// TwinCAT 3 PLC project MainPlc
// ProgramVersion: 3.1.4023.0
// libraries:
//   Tc2_Standard, * (Beckhoff Automation GmbH)
//   Tc2_System, * (Beckhoff Automation GmbH)
//   Tc3_Module, * (Beckhoff Automation GmbH)
// project tree:
//   App/Components/ fbDigitalSensor.TcPOU, fbPneumaticActuator.TcPOU, fbStepConveyor.TcPOU, stComponents.TcDUT, stPneumatics.TcDUT
//   App/Data/ fcEvalConitinuos.TcPOU, stContinuosValueData.TcDUT, stData.TcDUT
//   App/ enumMode.TcDUT (not stored), fbStation.TcPOU, MAIN.TcPOU
//   / IO.TcGVL, PlcTask.TcTTO (not stored)
//   ValueSimulation/ fbValueSimulation.TcPOU
// real-time tasks:
//   TASK PlcTask: cycle T#10ms, priority 20, ADS port 350
// I/O:
//   DEVICE Device 1 (EtherCAT) (disabled), AmsNetId 172.20.10.235.2.1
//     Term 1 (EK1100) [EK1100 EtherCAT Coupler (2A E-Bus)]
//       10A1 (EL1809) [EL1809 16Ch. Dig. Input 24V, 3ms]
//       10A2 (EL2809) [EL2809 16Ch. Dig. Output 24V, 0.5A]
// variable links:
//   MainPlc/MainPlc Instance <-> Device 1 (EtherCAT)/Term 1 (EK1100)/10A1 (EL1809)
//     PlcTask Inputs/IO.i10A1_CH{1..16} <-> Channel {1..16}/Input  (16 links)
//   MainPlc/MainPlc Instance <-> Device 1 (EtherCAT)/Term 1 (EK1100)/10A2 (EL2809)
//     PlcTask Outputs/IO.q10A2_CH{1..16} <-> Channel {1..16}/Output  (16 links)

// ---- App/Components/stComponents.TcDUT
{attribute wpf [Container(Layout.Tabs)]}
{attribute addProperty Name "<#Components#>"}
TYPE stComponents :
STRUCT		
	_pneumatics : stPneumatics;
	{attribute addProperty Name "<#Input step conveyor#> A4"}
	_inputConveyor : fbStepConveyor;	
	{attribute addProperty Name "<#Brick in the take-off position#>"}
	_BrickInTakeOffPosition : fbDigitalSensor;
	{attribute addProperty Name "<#Brick in the gripper#>"}
	_BrickInGripper : fbDigitalSensor;
	{attribute wpf [Container(Layout.Stack, "Measurement sensors")]}
	{attribute addProperty Name "<#Sensor dim X#>"}
	_X_DimSensor : REAL;
	{attribute addProperty Name "<#Sensor dim Y#>"}
	_Y_DimSensor : REAL;
	{attribute addProperty Name "<#Sensor dim Z#>"}
	_Z_DimSensor : REAL;
END_STRUCT
END_TYPE

// ---- App/Components/stPneumatics.TcDUT
{attribute wpf [Container(Layout.Stack)]}
{attribute addProperty Name "<#Pneumatics#>"}
TYPE stPneumatics :
STRUCT
	{attribute addProperty Name "<#Horizontal piston#> A1"}	
	_horizontalPiston : fbPneumaticActuator;
	{attribute addProperty Name "<#Vertical piston#> A2"}
	_verticalPiston : fbPneumaticActuator;
	{attribute addProperty Name "<#Gripper#> A3"}
	_gripper : fbPneumaticActuator;
	{attribute addProperty Name "<#Input end conveyor stopper#> A4"}
	_conveyorEndStopper : fbPneumaticActuator;		
END_STRUCT
END_TYPE

// ---- App/Data/stContinuosValueData.TcDUT
{attribute wpf [Container(Layout.Wrap)]}
{attribute wpf [Group(Layout.GroupBox)]}
TYPE stContinuosValueData :
STRUCT
	{attribute addProperty Name "<#Min#>"}
	Mininum : REAL;
	{attribute wpf [RenderIgnore("Control", "ShadowControl")]}
	{attribute addProperty Name "<#Aquired#>"}	
	Measured : REAL;
	{attribute addProperty Name "<#Max#>"}
	Maximum : REAL;	
END_STRUCT
END_TYPE

// ---- App/Data/stData.TcDUT
{attribute wpf [Container(Layout.Stack)]}
TYPE stData :
STRUCT
	{attribute addProperty Name "<#DimensionX#> [mm]"}			
	DimX : stContinuosValueData;
	{attribute addProperty Name "<#DimensionY#> [mm]"}
	DimY : stContinuosValueData;
	{attribute addProperty Name "<#DimensionZ#> [mm]"}
	DimZ : stContinuosValueData;
END_STRUCT
END_TYPE

// ---- IO.TcGVL
{attribute 'qualified_only'}
VAR_GLOBAL
	i10A1_CH1	AT %I* :BOOL;
	i10A1_CH2	AT %I* :BOOL;
	i10A1_CH3	AT %I* :BOOL;
	i10A1_CH4	AT %I* :BOOL;
	i10A1_CH5	AT %I* :BOOL;
	i10A1_CH6	AT %I* :BOOL;
	i10A1_CH7	AT %I* :BOOL;
	i10A1_CH8	AT %I* :BOOL;
	i10A1_CH9	AT %I* :BOOL;
	i10A1_CH10	AT %I* :BOOL;
	i10A1_CH11	AT %I* :BOOL;
	i10A1_CH12	AT %I* :BOOL;
	i10A1_CH13	AT %I* :BOOL;
	i10A1_CH14	AT %I* :BOOL;
	i10A1_CH15	AT %I* :BOOL;
	i10A1_CH16	AT %I* :BOOL;

	q10A2_CH1	AT %Q* :BOOL;
	q10A2_CH2	AT %Q* :BOOL;
	q10A2_CH3	AT %Q* :BOOL;
	q10A2_CH4	AT %Q* :BOOL;
	q10A2_CH5	AT %Q* :BOOL;
	q10A2_CH6	AT %Q* :BOOL;
	q10A2_CH7	AT %Q* :BOOL;
	q10A2_CH8	AT %Q* :BOOL;
	q10A2_CH9	AT %Q* :BOOL;
	q10A2_CH10	AT %Q* :BOOL;
	q10A2_CH11	AT %Q* :BOOL;
	q10A2_CH12	AT %Q* :BOOL;
	q10A2_CH13	AT %Q* :BOOL;
	q10A2_CH14	AT %Q* :BOOL;
	q10A2_CH15	AT %Q* :BOOL;
	q10A2_CH16	AT %Q* :BOOL;
END_VAR

// ---- App/Components/fbDigitalSensor.TcPOU
{attribute wpf [Container(Layout.Wrap)]}
{attribute wpf [Group(Layout.GroupBox)]}
FUNCTION_BLOCK fbDigitalSensor
VAR_INPUT
	{attribute 'hide'}
	Signal : BOOL;
END_VAR
VAR_OUTPUT
END_VAR
VAR
	{attribute wpf [Container(Layout.UniformGrid)]}
	{attribute addProperty Name "Value"}
	{attribute addProperty ToolTip "Sensor actual value"}
	Value : BOOL;
END_VAR

Value := Signal;

METHOD IsOff : BOOL
VAR_INPUT
END_VAR
Value := Signal;

IsOff := NOT Value;
END_METHOD

METHOD IsOn : BOOL
VAR_INPUT
END_VAR
Value := Signal;

IsOn := Value;
END_METHOD

END_FUNCTION_BLOCK

// ---- App/Components/fbPneumaticActuator.TcPOU
{attribute wpf [Container(Layout.Wrap)]}
{attribute wpf [Group(Layout.GroupBox)]}
FUNCTION_BLOCK fbPneumaticActuator
VAR_INPUT
	{attribute wpf [Container(Layout.Stack)]}	
	{attribute addProperty Name "Retracted"}
	{attribute addProperty ToolTip "Sensor indicating that the actuator is retracted"}
	inRetracted : BOOL;	
	{attribute addProperty Name "Extended"}
	{attribute addProperty ToolTip "Sensor indicating that the actuator is extended"}
	inExtended : BOOL;	
END_VAR
VAR_OUTPUT
	{attribute wpf [Container(Layout.Stack)]}
	{attribute addProperty Name "Retract"}
	{attribute addProperty ToolTip "Signal for retracting"}
	outRetract : BOOL;
	{attribute addProperty Name "Extend"}
	{attribute addProperty ToolTip "Signal for Extending"}
	outExtend : BOOL;
END_VAR
VAR
	{attribute wpf [Container(Layout.UniformGrid)]}
	{attribute addProperty Name "Retract command"}
	{attribute addProperty ToolTip "Executes retraction in manual mode"}
	_manualRetract : BOOL;
	{attribute addProperty Name "Extend command"}
	{attribute addProperty ToolTip "Executes extension in manual mode"}
	_manualExtend : BOOL;
END_VAR

METHOD Extend : BOOL
THIS^.outRetract := FALSE;
THIS^.outExtend := TRUE;

Extend := THIS^.inExtended;
END_METHOD

METHOD Manual
IF(THIS^._manualExtend AND_THEN THIS^.Extend()) THEN THIS^._manualExtend := FALSE; END_IF;
IF(THIS^._manualRetract AND_THEN THIS^.Retract()) THEN THIS^._manualRetract := FALSE; END_IF;

THIS^._manualExtend := FALSE;
THIS^._manualRetract := FALSE;
END_METHOD

METHOD Retract : BOOL
THIS^.outRetract := TRUE;
THIS^.outExtend := FALSE;

Retract := THIS^.inRetracted;
END_METHOD

END_FUNCTION_BLOCK

// ---- App/Components/fbStepConveyor.TcPOU
{attribute wpf [Container(Layout.Wrap)]}
{attribute wpf [Group(Layout.GroupBox)]}
FUNCTION_BLOCK fbStepConveyor
VAR_INPUT
	{attribute wpf [Container(Layout.Stack)]}	
	{attribute addProperty Name "Stop condition"}
	{attribute addProperty ToolTip "Signal that stops the conveyor"}
	inStop : BOOL;	
END_VAR
VAR_OUTPUT
	{attribute wpf [Container(Layout.Stack)]}
	{attribute addProperty Name "Move"}
	{attribute addProperty ToolTip "Signal for moving conveyor"}
	outMove : BOOL;
END_VAR
VAR
	{attribute wpf [Container(Layout.UniformGrid)]}
	{attribute addProperty Name "Move manual command"}
	{attribute addProperty ToolTip "Triggers movement in manual mode if possible"}
	_manualMove : BOOL;	
	{attribute 'hide'}
	_move : BOOL;	
	{attribute 'hide'}
	rtrg_inStop : R_TRIG;	
	{attribute 'hide'}
	_moveTimeout : TON;	
END_VAR

rtrg_inStop(CLK := inStop);

_moveTimeout(IN := THIS^._move, PT := T#500MS);

IF rtrg_inStop.Q OR _moveTimeout.Q THEN
	_move := FALSE;
END_IF


THIS^.outMove := _move;

METHOD Manual
IF THIS^._manualMove THEN THIS^._move := TRUE; END_IF;

THIS^._manualMove := FALSE;
END_METHOD

PROPERTY Run : BOOL
GET
END_GET
SET
_move := RUN;
END_SET
END_PROPERTY

END_FUNCTION_BLOCK

// ---- App/Data/fcEvalConitinuos.TcPOU
FUNCTION fcEvalConitinuos : BOOL
VAR_INPUT
	Val : REAL;
END_VAR
VAR_IN_OUT
	Data : stContinuosValueData;
END_VAR

Data.Measured := Val;
fcEvalConitinuos := (Data.Mininum <= Data.Measured AND Data.Measured <= Data.Maximum);

END_FUNCTION

// ---- App/fbStation.TcPOU
{attribute wpf [Container(Layout.Tabs)]}
{attribute addProperty Name "STATION 01"}
FUNCTION_BLOCK fbStation
VAR		
	{attribute wpf [Container(Layout.Stack)]}
	{attribute addProperty Name "<#Select mode#>"}
	_modeSelector : enumMode;
	{attribute clr [ReadOnly()]}
	{attribute addProperty Name "<#CurrentMode#>"}
	_modeCurrent : enumMode;
		
	{attribute addProperty Name "<#Step description#>"}
	_stepInfo : STRING[255];
	
	{attribute addProperty Name "<#Error description#>"}
	_errorInfo : STRING[255];
	
	{attribute addProperty Name "<#Components#>"}
	_components : stComponents;
	
	{attribute addProperty Name "<#Data#>"}
	_data : stData;
	
	_step : INT;

	_ground_done : BOOL;

	{attribute 'hide'}
	_errorTimer : TON;
	{attribute 'hide'}
	_lastStep : INT;
	
	{attribute 'hide'}
	_x : fbValueSimulation;
	{attribute 'hide'}
	_y : fbValueSimulation;
	{attribute 'hide'}
	_z : fbValueSimulation;

END_VAR

_components._pneumatics._horizontalPiston(inRetracted := IO.i10A1_CH1,
										  inExtended := IO.i10A1_CH2,
										  outRetract => IO.q10A2_CH1,
										  outExtend => IO.q10A2_CH2);
										  
_components._pneumatics._verticalPiston(inRetracted := IO.i10A1_CH3,
										  inExtended := IO.i10A1_CH4,
										  outRetract => IO.q10A2_CH3,
										  outExtend => IO.q10A2_CH4);										  

										  
_components._pneumatics._gripper(inRetracted := IO.i10A1_CH6,
										  inExtended := IO.i10A1_CH5,
										  outRetract => IO.q10A2_CH6,
										  outExtend => IO.q10A2_CH5);										  


_components._pneumatics._conveyorEndStopper(inRetracted := IO.i10A1_CH7,
										  inExtended := IO.i10A1_CH8,
										  outRetract => IO.q10A2_CH7,
										  outExtend => IO.q10A2_CH8);										  
										
_components._BrickInTakeOffPosition(Signal := IO.i10A1_CH9);
_components._BrickInGripper(Signal := IO.i10A1_CH10);

 _components._inputConveyor(inStop := _components._BrickInTakeOffPosition.IsOn(),
							outMove => IO.q10A2_CH9);


_x(MinValue:=247,MaxValue:=249);
_y(MinValue:=499,MaxValue:=501);
_z(MinValue:=248,MaxValue:=250);

_components._X_DimSensor := _x.Value;
_components._Y_DimSensor := _y.Value;
_components._Z_DimSensor := _z.Value;

							  
										  
_errorInfo := '';
_stepInfo := '';
//Reset step number in case of changing mode 
IF _modeCurrent <> _modeSelector THEN
	_step := 0;
END_IF

_modeCurrent := _modeSelector;

CASE _modeCurrent OF
	enumMode.Ground :
		GroundMode();
	enumMode.Automat :
		AutomatMode();
	enumMode.Manual:
		ManualMode();	
END_CASE

METHOD AutomatMode

VAR_INST
	_isOk : BOOL;	
END_VAR
IF NOT _ground_done THEN
	RETURN;
END_IF

_errorTimer(IN := _step = _lastStep, PT := T#10S);

IF(_errorTimer.Q) THEN
	_errorInfo := '<#This operation is taking way too long#>';
END_IF

_lastStep := _step;

CASE _step OF
	0:		
		_stepInfo := '<#Checking base position#>';		
//		_components._inputConveyor.Run := TRUE;

		IF(_components._pneumatics._verticalPiston.Retract() 
		AND_THEN _components._pneumatics._gripper.Extend() 
		AND_THEN _components._pneumatics._horizontalPiston.Retract()
		AND_THEN _components._pneumatics._conveyorEndStopper.Retract()) 
		THEN			
			_step := _step + 100;		
		END_IF
	100:
	   _stepInfo := '<#Measure the brick parameters.#>';
	   _isOk := fcEvalConitinuos(Val := _components._X_DimSensor, Data := _data.DimX)
				AND fcEvalConitinuos(Val := _components._Y_DimSensor, Data := _data.DimY)
				AND fcEvalConitinuos(Val := _components._Z_DimSensor, Data := _data.DimZ);
			IF _isOK THEN
				_step := 1000;		
			ELSE	
				_step := _step + 100;		
			END_IF;	
	200:
		_stepInfo := '<#Throwing away bad brick, openning end stoper.#>';
		IF(_components._pneumatics._conveyorEndStopper.Extend()) THEN
				_step := _step + 100;		
		END_IF;   
			
	300:
		_stepInfo := '<#Throwing away bad brick, moving conveyor.#>';
		_components._inputConveyor.Run := TRUE;
		IF(_components._BrickInTakeOffPosition.IsOff()) THEN
			_step := _step + 100;		
		END_IF;   

	400:
		_stepInfo := '<#Throwing away bad brick, moving conveyor.#>';
		_components._inputConveyor.Run := FALSE;
		IF(_components._BrickInTakeOffPosition.IsOn()) THEN
			_step := _step + 100;		
		END_IF;   

	500:
		_stepInfo := '<#Throwing away bad brick, closing end stoper.#>';
		IF(_components._pneumatics._conveyorEndStopper.Extend()) THEN
				_step := 1300;		
		END_IF;   
			
	1000:
		_stepInfo := '<#Take passed brick#>';
		IF(_components._pneumatics._verticalPiston.Extend() 
		AND_THEN _components._pneumatics._gripper.Retract())
		THEN
			_step := _step + 100;		
		END_IF;   
	1100:
		_stepInfo := '<#Move passed brick to output conveyor#>';
		IF(_components._pneumatics._verticalPiston.Retract()
		AND_THEN _components._pneumatics._horizontalPiston.Extend()) 		
		THEN			
			_components._inputConveyor.Run := TRUE;
			_step := _step + 100;		
		END_IF;		
	1200:
		_stepInfo := '<#Unload passed brick at the output conveyor#>';
		IF(_components._pneumatics._verticalPiston.Extend()
		AND_THEN _components._pneumatics._gripper.Extend()) THEN
			_step := _step + 100;		
		END_IF;			
	1300:		
		_stepInfo := '<#Stop step conveyor#>';
		_components._inputConveyor.Run := FALSE;
		_step := 0;	
END_CASE
END_METHOD

METHOD GroundMode : BOOL

_errorTimer(IN := _step = _lastStep, PT := T#3S);

IF(_errorTimer.Q) THEN
	_errorInfo := '<#This operation is taking way too long#>';
END_IF

_lastStep := _step;

CASE _step OF
	0:
		_ground_done := FALSE;
		_step := 10;
	10:		
		_stepInfo := '<#Moving everything to ground position#>';		
		IF(_components._pneumatics._verticalPiston.Retract() 
		AND_THEN _components._pneumatics._gripper.Extend() 
		AND_THEN _components._pneumatics._horizontalPiston.Retract()
		AND_THEN _components._pneumatics._conveyorEndStopper.Retract()) 
		THEN
			_step := 100;		
		END_IF
	100:
	   _stepInfo := '<#All in position ready to start#>';
	   _ground_done := TRUE;
	   _modeSelector := enumMode.None;
END_CASE
END_METHOD

METHOD ManualMode : BOOL
VAR_INPUT
END_VAR
_ground_done := FALSE;

_components._pneumatics._gripper.Manual();
_components._pneumatics._horizontalPiston.Manual();
_components._pneumatics._verticalPiston.Manual();
_components._pneumatics._conveyorEndStopper.Manual();
_components._inputConveyor.Manual();
END_METHOD

END_FUNCTION_BLOCK

// ---- ValueSimulation/fbValueSimulation.TcPOU
FUNCTION_BLOCK fbValueSimulation
VAR_INPUT
	MinValue : REAL;
	MaxValue : REAL;
END_VAR
VAR_OUTPUT
	Value : REAL;
END_VAR
VAR
	rn : DRAND;
END_VAR

rn();

Value := LREAL_TO_REAL(MinValue + rn.Num * (MaxValue-MinValue));

END_FUNCTION_BLOCK

// ---- App/MAIN.TcPOU
PROGRAM MAIN
VAR
	_station : fbStation;	
END_VAR

_station();

END_PROGRAM
